// TIA Portal V20 export
ORGANIZATION_BLOCK "CyclicInterrupt"   // OB30, LAD, CyclicInterrupt
{ S7_Optimized_Access := 'TRUE' }
// stored: SetENOAutomatically false
   VAR_INPUT
      Initial_Call : Bool;   // Initial call of this OB
      Event_Count : Int;   // Events discarded
   END_VAR
BEGIN

REGION Network 1
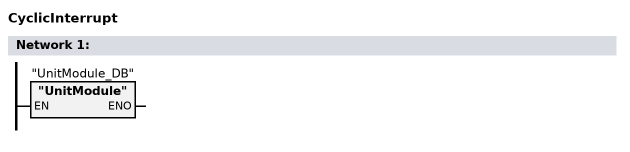
   RUNG wire#powerrail
      "UnitModule_DB"()
   END_RUNG
   // the same network as SCL:
   "UnitModule_DB"();   // "UnitModule"
END_REGION
END_ORGANIZATION_BLOCK
